{attribute 'qualified_only'}
{attribute 'strict'}
TYPE E_MachineStates :
(
	INIT 			:= 100,         // Initialization 
    CHECK_AIR_FLOW 	:= 110,         // Air Flow Verifying 
    SEAL_STAGES 	:= 130,         // Seal Stages/plates cycle 
    LEAK_TEST 		:= 140,         // Leak Test cycle 
	PRIME_SOLVENT	:= 150,			// Prime Solvents cycle 
    RECOVERY_PHASE 	:= 160,         // Recovery Cycle 
    WASHING_PHASE 	:= 170,         // Washing Cycle
    DRYING_PHASE 	:= 180,         // Drying Cycle
    POST_EXECUTION 	:= 190,         // Post Execution
	PAUSE_STATE		:= 200,			// Pause/Hold State
    ERROR_STATE 	:= 99           // Error State 
);
END_TYPE

(* stored: Version 1.1.0.1, ProductVersion 3.1.4024.15
   DUT E_MachineStates: Id {f3682b95-32d3-463a-bd62-ececb9b39ec1} *)
